(* IEC 61131-3 sources: 2026_Projet_YGO_ExcavatriceDragage/TOOLS/TEST_AUTO_CI/RESULTS/CYCLE/tests, 2 files *)

(* ---- test_fb_cycle.st ---- *)
SETUP
VAR
    FB : FB_Cycle;
    SampleCount : INT := 0;
END_VAR
END_SETUP

TEST 'Cycle : Enable=FALSE neutralise les commandes treuils/translation/benne'
    FB(Enable := FALSE, PowerContactorEngaged := TRUE, SampleCount := SampleCount);
    ASSERT_FALSE(FB.Ready, 'Ready doit etre FALSE sans Enable');
    ASSERT_FALSE(FB.WinchM1Cmd.StartStop, 'M1 coupe');
    ASSERT_FALSE(FB.WinchM2Cmd.StartStop, 'M2 coupe');
    ASSERT_FALSE(FB.TranslationCmd.Start, 'M3 coupe');
    ASSERT_FALSE(FB.BucketCmd.Open, 'Benne Open coupe');
    ASSERT_FALSE(FB.BucketCmd.Close, 'Benne Close coupe');
END_TEST

(* ---- test_fb_divesearch.st ---- *)
SETUP
VAR
    FB : FB_DiveSearch;
END_VAR
END_SETUP

TEST 'DiveSearch : Enable=FALSE neutralise les permis'
    FB(Enable := FALSE, PowerContactorEngaged := TRUE);
    ASSERT_FALSE(FB.Ready, 'Ready doit etre FALSE sans Enable');
    ASSERT_FALSE(FB.DescendPermit, 'DescendPermit doit etre FALSE');
    ASSERT_FALSE(FB.KoboldMeasureEnable, 'KoboldMeasureEnable doit etre FALSE');
END_TEST
